// Mitsubishi GX Works2 project: 240905_공급   PLC: Q03UDV

PROGRAM MAIN
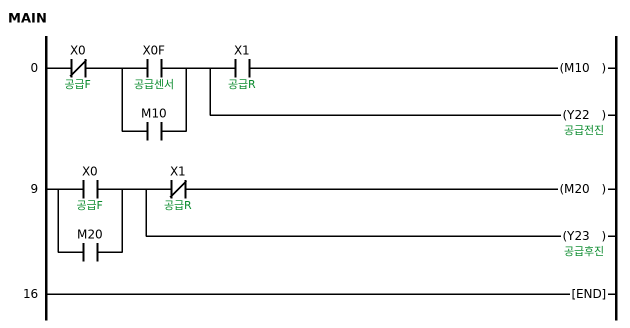
0     LDI     X0  ; 공급F
      LD      X0F  ; 공급센서
      OR      M10
      ANB
      MPS
      AND     X1  ; 공급R
      OUT     M10
      MPP
      OUT     Y22  ; 공급전진
9     LD      X0  ; 공급F
      OR      M20
      MPS
      ANI     X1  ; 공급R
      OUT     M20
      MPP
      OUT     Y23  ; 공급후진
16    END
END_PROGRAM
